// TIA Portal V15.1 export
// export: Created 2024-06-21T08:40:41.0843446Z, ExportSetting WithDefaults, DisplayName Totally Integrated Automation Portal, DisplayVersion V15.1 Update 5, DisplayName TIA Portal Openness, DisplayVersion V15.1 Update 5, DisplayName SINAMICS Startdrive Advanced, DisplayVersion V15.1, DisplayName G130, G150, S120, S150, SINAMICS MV, S210, DisplayVersion V15.1, DisplayName G110M, G120, G120C, G120D, G120P, DisplayVersion V15.1, DisplayName STEP 7 Professional, DisplayVersion V15.1 Update 5, DisplayName STEP 7 Safety, DisplayVersion V15.1, DisplayName WinCC Professional, DisplayVersion V15.1 Update 5, DisplayName SIMATIC Visualization Architect, DisplayVersion V15.1
DATA_BLOCK "_209000NCP01"   // DB1
{ S7_Optimized_Access := 'FALSE' }
AUTHOR : VCC
VERSION : 0.1
// stored: AutoNumber false, DBAccessibleFromOPCUA true, IsOnlyStoredInLoadMemory false, IsWriteProtectedInAS false
   VAR RETAIN
      SystemVar { ExternalAccessible := 'False'; ExternalVisible := 'False'; ExternalWritable := 'False'} : "AlarmBits";   // SystemVar Alarm Bits
      DiagPLCOverview { ExternalAccessible := 'False'; ExternalVisible := 'False'; ExternalWritable := 'False'} : "AlarmBits";   // DiagPLCOverview Alarm Bits
      ProdMode { ExternalAccessible := 'False'; ExternalVisible := 'False'; ExternalWritable := 'False'} : "AlarmBits";   // ProdMode Alarm Bits
      AE { ExternalAccessible := 'False'; ExternalVisible := 'False'; ExternalWritable := 'False'} : "AlarmBits";   // AE Alarm Bits
      AK { ExternalAccessible := 'False'; ExternalVisible := 'False'; ExternalWritable := 'False'} : "AlarmBits";   // AK Alarm Bits
      AS { ExternalAccessible := 'False'; ExternalVisible := 'False'; ExternalWritable := 'False'} : "AlarmBits";   // AS Alarm Bits
      Safety { ExternalAccessible := 'False'; ExternalVisible := 'False'; ExternalWritable := 'False'} : "AlarmBits";   // Safety Alarm Bits
      "209210ZS01" { ExternalAccessible := 'False'; ExternalVisible := 'False'; ExternalWritable := 'False'} : "AlarmBits";   // 209210ZS01 Alarm Bits
      "209220ZS01" { ExternalAccessible := 'False'; ExternalVisible := 'False'; ExternalWritable := 'False'} : "AlarmBits";   // 209220ZS01 Alarm Bits
      "209230ZS01" { ExternalAccessible := 'False'; ExternalVisible := 'False'; ExternalWritable := 'False'} : "AlarmBits";   // 209230ZS01 Alarm Bits
      Alarm { ExternalAccessible := 'False'; ExternalVisible := 'False'; ExternalWritable := 'False'} : "Alarm";   // Modes Alarm
      AlarmA { ExternalAccessible := 'False'; ExternalVisible := 'False'; ExternalWritable := 'False'} : Bool;   // Alarm A
      AlarmB { ExternalAccessible := 'False'; ExternalVisible := 'False'; ExternalWritable := 'False'} : Bool;   // Alarm B
      AlarmC { ExternalAccessible := 'False'; ExternalVisible := 'False'; ExternalWritable := 'False'} : Bool;   // Alarm C
      AlarmD { ExternalAccessible := 'False'; ExternalVisible := 'False'; ExternalWritable := 'False'} : Bool;   // Alarm D
      UpperLevelAlarmA { ExternalAccessible := 'False'; ExternalVisible := 'False'; ExternalWritable := 'False'} : Bool;   // AlarmA from this level , to connect to lower level LMode of your modezone
      UpperLevelAlarmB { ExternalAccessible := 'False'; ExternalVisible := 'False'; ExternalWritable := 'False'} : Bool;   // AlarmB from this level , to connect to lower level LMode of your modezone
      UpperLevelAlarmC { ExternalAccessible := 'False'; ExternalVisible := 'False'; ExternalWritable := 'False'} : Bool;   // AlarmC from this level , to connect to lower level LMode of your modezone
      UpperLevelAlarmD { ExternalAccessible := 'False'; ExternalVisible := 'False'; ExternalWritable := 'False'} : Bool;   // AlarmD from this level , to connect to lower level LMode of your modezone
      UpperLevelABCondition { ExternalAccessible := 'False'; ExternalVisible := 'False'; ExternalWritable := 'False'} : Bool;   // Alarm AB condition / Alarm D
      HMIAlarmReset { ExternalAccessible := 'False'; ExternalVisible := 'False'; ExternalWritable := 'False'} : Bool;   // Reset alarm from HMI
      HMIStart { ExternalAccessible := 'False'; ExternalVisible := 'False'; ExternalWritable := 'False'} : Bool;   // Start from HMI
      MorningShiftActive { ExternalAccessible := 'False'; ExternalVisible := 'False'; ExternalWritable := 'False'} : Bool;   // Morning shift is active
      EveningShiftActive { ExternalAccessible := 'False'; ExternalVisible := 'False'; ExternalWritable := 'False'} : Bool;   // Evening shift is active
      NightShiftActive { ExternalAccessible := 'False'; ExternalVisible := 'False'; ExternalWritable := 'False'} : Bool;   // Night shift is active
      NewShift { ExternalAccessible := 'False'; ExternalVisible := 'False'; ExternalWritable := 'False'} : Bool;   // New shift / Night shift is active
      ShiftOverview { ExternalAccessible := 'False'; ExternalVisible := 'False'; ExternalWritable := 'False'} : Struct   // Overview Active Shift
         MorningShift_Day1 { ExternalAccessible := 'False'; ExternalVisible := 'False'; ExternalWritable := 'False'} : Bool;   // Morning Shift of Day 1 (Monday)
         EveningShift_Day1 { ExternalAccessible := 'False'; ExternalVisible := 'False'; ExternalWritable := 'False'} : Bool;   // Evening Shift of Day 1 (Monday)
         NightShift_Day1 { ExternalAccessible := 'False'; ExternalVisible := 'False'; ExternalWritable := 'False'} : Bool;   // Night Shift of Day 1 (Monday-Tuesday)
         MorningShift_Day2 { ExternalAccessible := 'False'; ExternalVisible := 'False'; ExternalWritable := 'False'} : Bool;   // Morning Shift of Day 2 (Tuesday)
         EveningShift_Day2 { ExternalAccessible := 'False'; ExternalVisible := 'False'; ExternalWritable := 'False'} : Bool;   // Evening Shift of Day 2 (Tuesday)
         NightShift_Day2 { ExternalAccessible := 'False'; ExternalVisible := 'False'; ExternalWritable := 'False'} : Bool;   // Night Shift of Day 2 (Tuesday-Wednesday)
         MorningShift_Day3 { ExternalAccessible := 'False'; ExternalVisible := 'False'; ExternalWritable := 'False'} : Bool;   // Morning Shift of Day 3 (Wednesday)
         EveningShift_Day3 { ExternalAccessible := 'False'; ExternalVisible := 'False'; ExternalWritable := 'False'} : Bool;   // Evening Shift of Day 3 (Wednesday)
         NightShift_Day3 { ExternalAccessible := 'False'; ExternalVisible := 'False'; ExternalWritable := 'False'} : Bool;   // night Shift of Day 3 (Wednesday-Thursday)
         MorningShift_Day4 { ExternalAccessible := 'False'; ExternalVisible := 'False'; ExternalWritable := 'False'} : Bool;   // Morning Shift of Day 4 (Thursday)
         EveningShift_Day4 { ExternalAccessible := 'False'; ExternalVisible := 'False'; ExternalWritable := 'False'} : Bool;   // Evening Shift of Day 4 (Thursday)
         NightShift_Day4 { ExternalAccessible := 'False'; ExternalVisible := 'False'; ExternalWritable := 'False'} : Bool;   // Night Shift of Day 4 (Thursday-Friday)
         MorningShift_Day5 { ExternalAccessible := 'False'; ExternalVisible := 'False'; ExternalWritable := 'False'} : Bool;   // Morning Shift of Day 5 (Friday)
         EveningShift_Day5 { ExternalAccessible := 'False'; ExternalVisible := 'False'; ExternalWritable := 'False'} : Bool;   // Evening Shift of Day 5 (Friday)
         NightShift_Day5 { ExternalAccessible := 'False'; ExternalVisible := 'False'; ExternalWritable := 'False'} : Bool;   // Night Shift of Day 5 (Friday-Saturday)
         MorningShift_Day6 { ExternalAccessible := 'False'; ExternalVisible := 'False'; ExternalWritable := 'False'} : Bool;   // Morning Shift of Day 6 (Saturday)
         EveningShift_Day6 { ExternalAccessible := 'False'; ExternalVisible := 'False'; ExternalWritable := 'False'} : Bool;   // Evening Shift of Day 6 (Saturday)
         NightShift_Day6 { ExternalAccessible := 'False'; ExternalVisible := 'False'; ExternalWritable := 'False'} : Bool;   // Night Shift of Day 6 (Saturday-Sunday)
         MorningShift_Day7 { ExternalAccessible := 'False'; ExternalVisible := 'False'; ExternalWritable := 'False'} : Bool;   // Morning Shift of Day 7 (Sunday)
         EveningShift_Day7 { ExternalAccessible := 'False'; ExternalVisible := 'False'; ExternalWritable := 'False'} : Bool;   // Evening Shift of Day 7 (Sunday)
         NightShift_Day7 { ExternalAccessible := 'False'; ExternalVisible := 'False'; ExternalWritable := 'False'} : Bool;   // night Shift of Day 7 (Sunday-Monday)
      END_STRUCT;
      AlarmABCondition { ExternalAccessible := 'False'; ExternalVisible := 'False'; ExternalWritable := 'False'} : Bool;   // Alarm AB condition
      GeneralStart { ExternalAccessible := 'False'; ExternalVisible := 'False'; ExternalWritable := 'False'} : Bool;   // Summary of all start buttons
      GeneralStop { ExternalAccessible := 'False'; ExternalVisible := 'False'; ExternalWritable := 'False'} : Bool;   // Summary of all stop buttons
      GeneralReset { ExternalAccessible := 'False'; ExternalVisible := 'False'; ExternalWritable := 'False'} : Bool;   // Summary of all alarm reset buttons
      SumAlarmResetPassivationPB { ExternalAccessible := 'False'; ExternalVisible := 'False'; ExternalWritable := 'False'} : Bool;   // Summary of all alarm reset Passivation buttons
      SumLampentest { ExternalAccessible := 'False'; ExternalVisible := 'False'; ExternalWritable := 'False'} : Bool;   // Summary of all lampentest buttons
      H_DiagPLCOverviewIAnim : Word;   // For animation of icon
      H_AEIAnim : Word;   // For animation of icon
      H_AKIAnim : Word;   // For animation of icon
      H_ASIAnim : Word;   // For animation of icon
      H_SafetyIAnim : Word;   // For animation of icon
      H_209210ZS01IAnim : Word;   // For animation of icon
      H_209220ZS01IAnim : Word;   // For animation of icon
      H_209230ZS01IAnim : Word;   // For animation of icon
      H_IAnim : Word;   // For animation of icon
      H_Anim : Word;   // Animation
      H_Anim2 : Word;   // Animation
      H_DBnr : Int;   // DB number
      H_HMICmd : Word;   // HMI command
      H_ActiveShiftIAnim : Word;   // For animation of icon
      H_LVccLibVersion : String;   // LVccLibVersion
      H : Struct   // For animation
         "SystemVarS7-1500" : "H_SystemVarS7-1500";   // For animation
      END_STRUCT;
      H_HMI : Struct   // For animation of icon
         "SystemVarS7-1500" : "H_HMI";   // For animation of icon
      END_STRUCT;
      WeekendModeSel { ExternalAccessible := 'False'; ExternalVisible := 'False'; ExternalWritable := 'False'} : Bool;   // Global Production Modes - Weekend mode selected
      WeekendMode { ExternalAccessible := 'False'; ExternalVisible := 'False'; ExternalWritable := 'False'} : Bool;   // Global Production Modes - Weekend mode active
      MaintModeSel { ExternalAccessible := 'False'; ExternalVisible := 'False'; ExternalWritable := 'False'} : Bool;   // Global Production Modes - Maintenance mode selected
      MaintMode { ExternalAccessible := 'False'; ExternalVisible := 'False'; ExternalWritable := 'False'} : Bool;   // Global Production Modes - Maintenance mode active
      ProdStopModeSel { ExternalAccessible := 'False'; ExternalVisible := 'False'; ExternalWritable := 'False'} : Bool;   // Global Production Modes - Production stop mode selected
      ProdStopMode { ExternalAccessible := 'False'; ExternalVisible := 'False'; ExternalWritable := 'False'} : Bool;   // Global Production Modes - Production stop mode active
      AnyProdModeSel { ExternalAccessible := 'False'; ExternalVisible := 'False'; ExternalWritable := 'False'} : Bool;   // Global Production Modes - Any production mode selected
      AnyProdModeAct { ExternalAccessible := 'False'; ExternalVisible := 'False'; ExternalWritable := 'False'} : Bool;   // Global Production Modes - Any production mode active
      ProcProdMode { ExternalAccessible := 'False'; ExternalVisible := 'False'; ExternalWritable := 'False'} : Word;   // Global Production Modes - Production modes
      TimerSumAlarmResetPB { ExternalAccessible := 'False'; ExternalVisible := 'False'; ExternalWritable := 'False'} : TOF_TIME;   // Timer
      TimerSumAlarmResetPassivationPB { ExternalAccessible := 'False'; ExternalVisible := 'False'; ExternalWritable := 'False'} : TOF_TIME;   // Timer
      TimerSumAlarmStartPB { ExternalAccessible := 'False'; ExternalVisible := 'False'; ExternalWritable := 'False'} : TOF_TIME;   // Timer
   END_VAR
BEGIN
END_DATA_BLOCK
